RoboDK station: RobotVision.rdk

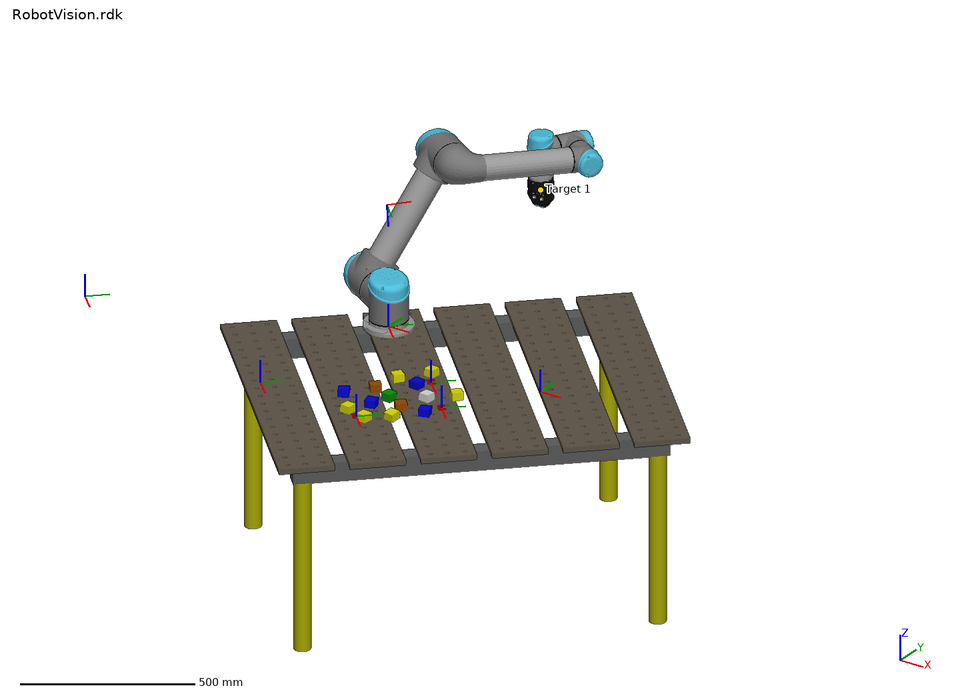
[picture v0: the station drawn from its stored meshes, robots at their saved joint values, targets as dots, program paths as lines]
Station TEST_DK (saved by RoboDK 5.6.0). Poses are relative to the parent item; angles as X-Y-Z fixed-axis rotations.
  - frame UR5 Base at (-500, 0, 0) mm
    - robot UR5: 6 axes
        modified DH rows (alpha deg, a mm, theta deg, d mm): 0, 0, 0, 89.2; 90, 0, 180, 0; 0, 425, 0, 0; 0, 392, 0, 109.3; -90, 0, 0, 94.75; 90, 0, 0, 82.5
        joint limits [-360, -360, -360, -360, -360, -360] to [360, 360, 360, 360, 360, 360]; home [0, -90, -90, 0, 90, 0]; saved at [-120.576, -56.937, -296.783, -276.28, 90, -30.576]
      - robot RobotiQ 2F-85 Gripper (Mechanism) (model RobotiQ 2F85): 1 axes, payload 5 kg
          joint limits [0] to [85]; home [85]; saved at [85]
        - tool Tool 1, TCP at (0, 0, 40) mm
    - target Target 1 (Cartesian target) at (173.85, 509.12, 280) mm, rotated rx -180 ry 0 rz 180 deg; joints [-56.79, -168.493, -261.575, -199.931, 90, 78.21] of UR5
  - frame Camera_Frame at (-208.51, -423.14, 637.3) mm, rotated rx -176.46 ry -3.53 rz 44.89 deg
    - camera Camera
  - frame Frame 4 at (100, -100, 0) mm
  - object Table 1200x1000mm (Welding) at (-140.01, -182.09, 0) mm, rotated rx 0 ry 0 rz -135 deg, size 1193.8 x 965.2 x 609.6 mm, geometry from Table-1200x1000mm-Welding.sld
  - frame Frame 4 at (-500, 0, 0) mm, rotated rx 0 ry 0 rz -45 deg
  - frame RED DOTIII at (-191.7, -227.69, 0) mm, rotated rx 0 ry 0 rz -45 deg
  - frame Figure at (-590, -510, 0) mm, rotated rx 0 ry 0 rz -45 deg
  - folder Cubes
    - object reddot2 at (-261, -528.92, -30) mm, rotated rx 0 ry 0 rz -45 deg, size 32 x 24 x 32 mm, geometry from Duplo.STL
    - object reddot3 at (-211.5, -224.86, -30) mm, rotated rx 0 ry 0 rz -45 deg, size 32 x 24 x 32 mm, geometry from Duplo.STL
    - object reddot1 at (-91.15, -345.21, -30) mm, rotated rx 0 ry 0 rz -45 deg, size 32 x 24 x 32 mm, geometry from Duplo.STL
    - object yellow5 at (-294.92, -533.73, 0) mm, rotated rx 90 ry 0 rz 85 deg, size 32 x 24 x 32 mm, geometry from Duplo.STL
    - object yellow3 at (-274.92, -293.73, 0) mm, rotated rx 90 ry 0 rz 145 deg, size 32 x 24 x 32 mm, geometry from Duplo.STL
    - object yellow1 at (-234.92, -203.73, 0) mm, rotated rx 90 ry 0 rz 85 deg, size 32 x 24 x 32 mm, geometry from Duplo.STL
    - object blue2 at (-223.64, -293.35, 0) mm, rotated rx 90 ry 0 rz 85 deg, size 32 x 24 x 32 mm, geometry from Duplo.STL
    - object white at (-153.64, -343.35, 0) mm, rotated rx 90 ry 0 rz 85 deg, size 32 x 24 x 32 mm, geometry from Duplo.STL
    - object blue4 at (-353.64, -463.35, 0) mm, rotated rx 90 ry 0 rz 120 deg, size 32 x 24 x 32 mm, geometry from Duplo.STL
    - object orange1 at (-314.92, -363.73, 0) mm, rotated rx 90 ry 0 rz 45 deg, size 32 x 24 x 32 mm, geometry from Duplo.STL
    - object yellow2 at (-94.92, -273.73, 0) mm, rotated rx 90 ry 0 rz 50 deg, size 32 x 24 x 32 mm, geometry from Duplo.STL
    - object orange2 at (-163, -443, 0) mm, rotated rx 90 ry 0 rz 135.68 deg, size 32 x 24 x 32 mm, geometry from Duplo.STL
    - object blue1 at (-253.64, -473.35, 0) mm, rotated rx 90 ry 0 rz 105 deg, size 32 x 24 x 32 mm, geometry from Duplo.STL
    - object green at (-243.64, -403.35, 0) mm, rotated rx 90 ry 0 rz 85 deg, size 32 x 24 x 32 mm, geometry from Duplo.STL
    - object yellow6 at (-163, -503, 0) mm, rotated rx 90 ry -7.08 rz 85 deg, size 32 x 24 x 32 mm, geometry from Duplo.STL
    - object yellow4 at (-224.92, -553.73, 0) mm, rotated rx 90 ry 0 rz 85 deg, size 32 x 24 x 32 mm, geometry from Duplo.STL
    - object blue3 at (-93.64, -433.35, 0) mm, rotated rx 90 ry 0 rz 110 deg, size 32 x 24 x 32 mm, geometry from Duplo.STL
  - frame StartingPosition at (-1087.57, -672.84, 200) mm, rotated rx 0 ry 0 rz -45 deg
  - frame RED DOT II at (-71.35, -348.04, 0) mm, rotated rx 0 ry 0 rz -45 deg
  - frame RED DOT I at (-241.2, -531.74, 0) mm, rotated rx 0 ry 0 rz -45 deg
  - program Replace_Objects2 (1 instructions, listed below)

--- program Replace_Objects2 (robot UR5) ---
  Replace objects
